Staubli VAL3: onStart.pgx

public program onStart(string& x_sItem[])
  local num i
  local string l_sType
  local string l_sPath
begin
  call language2:getLanguage(l_sPath)
  if l_sPath!=language2:libPath()+"/"+saveData:language
    // set language
    call language2:setLanguage(language2:libPath()+"/"+saveData:language)
  endIf
  // reset all the pallet
  call reset()
end
